(* PLC project FolderModule, Beckhoff Automation GmbH TwinCAT PLC Control 3.5.1.0 *)
(* stored: creationDateTime 2013-03-04T12:57:29.363091, modificationDateTime 2013-03-04T12:57:29.363091 *)

(* Automatic generated code. Do not change. Use Code generator instead. *)
PROGRAM ForcingLayer
  VAR
    In_EmergencyStop_Mapping AT %I* : BOOL;  (* In_EmergencyStop *)
    In_MotorFailure_Mapping AT %I* : BOOL;  (* In_MotorFailure *)
    Out_MotorTls_Mapping AT %Q* : BOOL;  (* Out_MotorTls *)
  END_VAR
  VAR
    EnableForcing : BOOL;
    In_EmergencyStop_EnableForcing : BOOL;
    In_EmergencyStop_Forcing : BOOL;
    In_MotorFailure_EnableForcing : BOOL;
    In_MotorFailure_Forcing : BOOL;
    Out_MotorTls_EnableForcing : BOOL;
    Out_MotorTls_Forcing : BOOL;
  END_VAR

            // Automatic generated code. Do not change. Use Code generator instead.
          

ACTION ForceInputs:
                // Automatic generated code. Do not change. Use Code generator instead.

IF EnableForcing THEN
	
	// In_EmergencyStop
	IF In_EmergencyStop_EnableForcing THEN
		In_EmergencyStop := In_EmergencyStop_ForceValue;
	ELSE
		In_EmergencyStop := In_EmergencyStop_Mapping;
	END_IF

	// In_MotorFailure
	IF In_MotorFailure_EnableForcing THEN
		In_MotorFailure := In_MotorFailure_ForceValue;
	ELSE
		In_MotorFailure := In_MotorFailure_Mapping;
	END_IF
	
ELSE
	
	In_EmergencyStop := In_EmergencyStop_Mapping;
	In_MotorFailure := In_MotorFailure_Mapping;
	
END_IF
              
END_ACTION

ACTION ForceOutputs:
                // Automatic generated code. Do not change. Use Code generator instead.

IF EnableForcing THEN
	
	// Out_MotorTls
	IF Out_MotorTls_EnableForcing THEN
		Out_MotorTls := Out_MotorTls_ForceValue;
	ELSE
		Out_MotorTls := Out_MotorTls_Mapping;
	END_IF

ELSE
	
	Out_MotorTls := Out_MotorTls_Mapping;
	
END_IF
              
END_ACTION
END_PROGRAM
